// TwinCAT 3 PLC project PLC2
// ProgramVersion: 3.1.4024.0
// libraries:
//   Tc2_DataExchange, * (Beckhoff Automation GmbH)
//   Tc2_Standard, * (Beckhoff Automation GmbH)
//   Tc2_System, * (Beckhoff Automation GmbH)
//   Tc3_Module, * (Beckhoff Automation GmbH)
// project tree:
//   DUTs/ ST_StorageSlot.TcDUT
//   / PlcTask.TcTTO
//   POUs/ FB_Example1.TcPOU, FB_Example2.TcPOU, FB_WriteExampl1.TcPOU, MAIN.TcPOU
// (motion and I/O tree: see PLC project practice_tdd)
// real-time tasks:
//   TASK PlcTask: cycle T#10ms, priority 20, ADS port 350
//   TASK PlcTask1: cycle T#10ms, priority 21, ADS port 351
//   TASK PlcTask2: cycle T#10ms, priority 22, ADS port 352

CONFIGURATION PLC2
    RESOURCE PLC ON TwinCAT3
        TASK PlcTask(INTERVAL := T#10ms, PRIORITY := 22);
        PROGRAM MAIN WITH PlcTask : MAIN;
    END_RESOURCE
END_CONFIGURATION

// ---- DUTs/ST_StorageSlot.TcDUT
TYPE ST_StorageSlot :
STRUCT
	nStorageId : INT;
	nStorageName : STRING;
	bMaintanence : BOOL;
END_STRUCT
END_TYPE

// ---- POUs/MAIN.TcPOU
PROGRAM MAIN
VAR
	
    bExecute1    : BOOL := FALSE;
	bExecute2    : BOOL := FALSE;
    nReadValue  : INT;           
    bBusy       : BOOL;
    bError      : BOOL;
    nErrId      : UDINT;
	sSymbol     : STRING := 'GVL_Config.nNumber';
	fbAdsRead1   : ADSRDWRTEX;
	fbAdsRead2   : ADSREAD;
	hVariable   : DWORD;
	
	fbRead1 : FB_Example1;
	fbRead2 : FB_Example2;
	fbWrite1 : FB_WriteExampl1;
	

END_VAR

IF bExecute1 THEN
	
	fbAdsRead1(
            NETID:= '', 
            PORT:= 852, 
            IDXGRP:= 16#F003,     
            IDXOFFS:= 0, 
            READLEN:= SIZEOF(hVariable),
			WRITELEN := INT_TO_UDINT(LEN(sSymbol)),
            SRCADDR:= ADR(sSymbol), 
            DESTADDR:= ADR(hVariable), 
            WRTRD:= TRUE, 
            BUSY => bBusy, ERR => bError, ERRID => nErrId);	
END_IF

IF bExecute2 THEN
	fbAdsRead2(
	NETID:= '', 
	PORT:= 852, 
	IDXGRP:= 16#F005 , 
	IDXOFFS:= hVariable, 
	LEN:= SIZEOF(nReadValue), 
	DESTADDR:= ADR(nReadValue), 
	READ:= bExecute2 , 
	BUSY => bBusy, 
	ERR => bError, 
	ERRID => nErrId);	
END_IF
fbRead1();
fbRead2();
fbWrite1();

END_PROGRAM

// ---- POUs/FB_Example1.TcPOU
FUNCTION_BLOCK FB_Example1

VAR
	fbRead1     :  FB_ReadAdsSymByName;
	bEnable     : BOOL;
	sSymbol     : STRING := 'GVL_Config.nNumber';
	nReadValue  : INT;
	eComMode    :  E_AdsComMode := eAdsComModeFastCom;
	bBusy       : BOOL;
    bError      : BOOL;
    nErrId      : UDINT;
	bExecute: BOOL;
	fbTimer : TON := (PT := T#100MS); // Adjust the speed here
END_VAR


fbTimer(IN := NOT fbTimer.Q); // This creates a self-resetting pulse

IF fbTimer.Q THEN
    bEnable := TRUE; // Trigger your FB_ReadAdsSymByName
END_IF

	fbRead1(
	bRead:= bEnable, 
	sNetId:= '', 
	nPort:= 852, 
	sVarName:= sSymbol, 
	nDestAddr:= ADR(nReadValue), 
	nLen:= SIZEOF(nReadValue), 
	tTimeout:= , 
	eComMode:= eComMode, 
	bClearOnError:= , 
	bBusy=> bBusy, 
	bError=> bError, 
	nErrorId=> nErrId);
bEnable := FALSE;

END_FUNCTION_BLOCK

// ---- POUs/FB_Example2.TcPOU
FUNCTION_BLOCK FB_Example2

VAR
	fbRead1     :  FB_ReadAdsSymByName;
	bEnable     : BOOL;
	sSymbol     : STRING := 'GVL_Config.arrRack[1]';
	stStorageSlot : ST_StorageSlot;
	eComMode    :  E_AdsComMode := eAdsComModeFastCom;
	bBusy       : BOOL;
    bError      : BOOL;
    nErrId      : UDINT;
	bExecute: BOOL;
	fbTimer : TON := (PT := T#100MS); // Adjust the speed here
END_VAR


fbTimer(IN := NOT fbTimer.Q); // This creates a self-resetting pulse

IF fbTimer.Q THEN
    bEnable := TRUE; // Trigger your FB_ReadAdsSymByName
END_IF

	fbRead1(
	bRead:= bEnable, 
	sNetId:= '', 
	nPort:= 852, 
	sVarName:= sSymbol, 
	nDestAddr:= ADR(stStorageSlot), 
	nLen:= SIZEOF(stStorageSlot), 
	tTimeout:= , 
	eComMode:= eComMode,
	bBusy=> bBusy, 
	bError=> bError, 
	nErrorId=> nErrId);
bEnable := FALSE;

END_FUNCTION_BLOCK

// ---- POUs/FB_WriteExampl1.TcPOU
FUNCTION_BLOCK FB_WriteExampl1

VAR
	fbRead1     :  FB_WriteAdsSymByName;
	bEnable     : BOOL;
	sSymbol     : STRING := 'GVL_Config.nNumber';
	nReadValue  : INT := 200;
	eComMode    :  E_AdsComMode := eAdsComModeSecureCom;
	bBusy       : BOOL;
    bError      : BOOL;
    nErrId      : UDINT;
	bExecute: BOOL;
	fbTimer : TON := (PT := T#100MS); // Adjust the speed here
END_VAR


	fbRead1(
	bWrite:= bEnable, 
	sNetId:= '', 
	nPort:= 852, 
	sVarName:= sSymbol, 
	nSrcAddr:= ADR(nReadValue), 
	nLen:= SIZEOF(nReadValue), 
	tTimeout:= , 
	eComMode:= eComMode,  
	bBusy=> bBusy, 
	bError=> bError, 
	nErrorId=> nErrId);
bEnable := FALSE;

END_FUNCTION_BLOCK
